PROGRAM PRG_Stats
VAR_INPUT
    nSample : DINT;
END_VAR
VAR_OUTPUT
    nMax : DINT;
END_VAR
VAR
    nCalls : UDINT;
    nSum : DINT;
END_VAR

nCalls := nCalls + 1;
Accumulate(nSample);

METHOD PRIVATE Accumulate
VAR_INPUT
    nValue : DINT;
END_VAR
nSum := nSum + nValue;
IF nValue > nMax THEN
    nMax := nValue;
END_IF
END_METHOD

PROPERTY Mean : DINT
GET
IF nCalls > 0 THEN
    Mean := nSum / UDINT_TO_DINT(nCalls);
END_IF
END_GET
END_PROPERTY

ACTION Clear:
nCalls := 0;
nSum := 0;
nMax := 0;
END_ACTION

END_PROGRAM

(* stored: Version 1.1.0.1, ProductVersion 3.1.4024.12
   POU PRG_Stats: Id {5f1c2d9e-0a6b-4c11-9d3e-7a1b2c3d4e90}, SpecialFunc None
   Method Accumulate: Id {5f1c2d9e-0a6b-4c11-9d3e-7a1b2c3d4e91}
   Property Mean: Id {5f1c2d9e-0a6b-4c11-9d3e-7a1b2c3d4e92}
   Get Get: Id {5f1c2d9e-0a6b-4c11-9d3e-7a1b2c3d4e93}
   Action Clear: Id {5f1c2d9e-0a6b-4c11-9d3e-7a1b2c3d4e94} *)
